(* PLC project OOP_Curso, Beckhoff Automation GmbH TwinCAT PLC Control 3.5.13.21 *)
(* stored: creationDateTime 2023-06-10T12:40:30.8169703, modificationDateTime 2023-06-10T12:40:30.8169703 *)

{attribute 'enable_dynamic_creation'}
TYPE ST_Estructura :
STRUCT
	dato1 : LWORD;
	dato2: DINT;
	dato3: SINT;
END_STRUCT
END_TYPE

PROGRAM _17_Otros_Operadores
VAR
	pEstructura : POINTER TO ST_Estructura;
	struNew     : BOOL;
END_VAR
VAR
	pSTRING  : POINTER TO STRING;
	bNew     : BOOL;
END_VAR	
VAR CONSTANT
	cLength  : UINT := 150;
END_VAR
VAR
	StruDelete  : BOOL;
END_VAR

            // Ejemplos de los Operadores __NEW y  __DELETE
IF struNew AND (pEstructura = 0) THEN
	pEstructura := __NEW(ST_Estructura);	
	struNew := FALSE;
END_IF

IF bNew THEN
    pSTRING := __NEW(BYTE, cLength);
    bNew    := FALSE;
END_IF

IF StruDelete THEN
	 __DELETE(pEstructura);	
	 __DELETE(pSTRING);	
	StruDelete := FALSE;
END_IF
          
END_PROGRAM
